  thread runBalayage():
    while (True):
        global ctrl_frequency=350.0
        global weave_frequency=1.2
        global amplitude=0.003
        global cycle_duration=(ctrl_frequency / weave_frequency)
        global pi=3.14159
        global offset=[0.0, 0.0, 0.0, 0.0, 0.0, 0.0]
        global i=0
        path_offset_enable()
        global alpha=0.1
        path_offset_set_alpha_filter(alpha)

        while (True):
          fct_set_offset()
          path_offset_set(offset, 2)
          global i=i+1
          sync()
        end
      end

  end

  def fct_activerBalayage(p_start, p_stop):

      fct_determineAxeBalayage(p_start,p_stop)
      global thr_runBalayage = run runBalayage()

  end

  def fct_desactiverBalayage():

      kill thr_runBalayage

  end
  $ 73 "Script: fcts_ralentir_fin_ligne.script"
  def fct_calcul_point_inter(p_debut,p_fin):

      local p_inter = p_fin

      local poucentage = 0.95
      local inc = 0
      local vecteur_global = p[0,0,0,0,0,0]
      local vecteur_reduit = p[0,0,0,0,0,0]

      while (inc < 6):   #a valider avec d'autres tests (peut etre faire une moyenne)
          vecteur_global[inc] = p_fin[inc] - p_debut[inc]
          vecteur_reduit[inc] = vecteur_global[inc]*poucentage
          p_inter[inc] = p_debut[inc] + vecteur_reduit[inc]
          inc = inc +1
      end

      return p_inter
    end


  $ 351 "Thread_1"
  thread Thread_1():
    while (True):
      $ 352 "Test_Ordre_Marche"
      $ 353 "If Test_Ordre_Mar≟ True "
      if (Test_Ordre_Mar ==   True  ):
        $ 354 "If config_d ≟ 1  or  config_g ≟ 1"
        if (config_d  ==  1   or   config_g  ==  1):
          $ 355 "Set Ordre_Marche=On"
          set_standard_digital_out(0, True)
          $ 356 "Wait: 0.5"
          sleep(0.5)
          $ 357 "If Reponse_Ordre≟ False "
          if (get_standard_digital_in(4) ==   False  ):
            $ 358 "'Si aucune reponse n'a etait recue, arret du programme'"
            # 'Si aucune reponse n'a etait recue, arret du programme'
            $ 359 "close_popup()"
            close_popup()
            $ 360 "Popup: Defaut : L'Ordre marche a ete coupe ( le poste est peu-etre eteint ) "
            popup("Defaut : L'Ordre marche a ete coupe ( le poste est peu-etre eteint ) ", "Error", False, True, blocking=False)
            halt
          end
          $ 361 "Test_Ordre_Mar≔ False "
          global Test_Ordre_Mar=  False
          $ 362 "sync()"
          sync()
        end
      end
      $ 363 "Erreur ordre marche pendant utilisation"
      $ 364 "If Arc_On≟ True   and Reponse_Arc≟ True  and Reponse_Ordre≟ False "
      if (get_standard_digital_out(1) ==   True     and  get_standard_digital_in(5) ==   True    and  get_standard_digital_in(4) ==   False  ):
        $ 365 "'Test pour savoir si ordre marche a ete coupe pendant utilisation'"
        # 'Test pour savoir si ordre marche a ete coupe pendant utilisation'
        $ 366 "close_popup()"
        close_popup()
        $ 367 "Popup: Defaut : Mise sous puissance coupee pendant la trajectoire"
        popup("Defaut : Mise sous puissance coupee pendant la trajectoire", "Error", False, True, blocking=False)
        halt
      end
      $ 368 "sync()"
      sync()
    end
  end
  threadId_Thread_1 = run Thread_1()
  $ 369 "Thread_2"
  thread Thread_2():
    while (True):
      $ 370 "mode_soudure"
      $ 371 "If Mode_soudure ≟  True "
      if (get_configurable_digital_in(3)  ==    True  ):
        $ 372 "If Mode_soudure≟ True  and soudure_on ≟ True "
        if (get_configurable_digital_in(3) ==   True    and  soudure_on  ==   True  ):
          $ 373 "fin_soud≔0"
          global fin_soud=0
          $ 374 "Test_Ordre_Mar≔ True "
          global Test_Ordre_Mar=  True
          $ 375 "Test_Job≔ True "
          global Test_Job=  True
          $ 376 "Wait Test_Ordre_Mar≟ False "
          while (not(Test_Ordre_Mar ==   False  )):
            sync()
          end
          $ 377 "Wait Test_Job≟ False "
          while (not(Test_Job ==   False  )):
            sync()
          end
          $ 378 "Set Arc_On=On"
          set_standard_digital_out(1, True)
          $ 379 "Test_Gaz≔ True "
          global Test_Gaz=  True
          $ 380 "'Test_Gaz permet de faire un appel dans le thread pour tester l'arriver gaz'"
          # 'Test_Gaz permet de faire un appel dans le thread pour tester l'arriver gaz'
          $ 381 "Wait Valide_Gaz≟ True "
          while (not(Valide_Gaz ==   True  )):
            sync()
          end
          $ 382 "'Valide_Gaz permet  de connaitre quand le traitement de l'arriver gaz est terminer ans le thread.'"
          # 'Valide_Gaz permet  de connaitre quand le traitement de l'arriver gaz est terminer ans le thread.'
        else:
          $ 383 "ElseIf Mode_soudure ≟ True  and soudure_on ≟ False "
          if (get_configurable_digital_in(3)  ==   True    and  soudure_on  ==   False  ):
            $ 384 "'Attente post debit gaz'"
            # 'Attente post debit gaz'
            $ 385 "Set Arc_On=Off"
            set_standard_digital_out(1, False)
            $ 386 "Test_Gaz≔ False "
            global Test_Gaz=  False
            $ 387 "Loop Reponse_Arc ≟ 1"
            while (get_standard_digital_in(5)  ==  1):
              $ 388 "fin_soud≔0"
              global fin_soud=0
              $ 389 "sync()"
              sync()
            end
            $ 390 "fin_soud≔1"
            global fin_soud=1
          end
        end
      end
      $ 391 "sync()"
      sync()
    end
  end
  threadId_Thread_2 = run Thread_2()
  $ 392 "Thread_3"
  thread Thread_3():
    while (True):
      $ 393 "led_cobot_2"
      $ 394 "If led_cobot ≟ True "
      if (led_cobot  ==   True  ):
        $ 395 "If valider_bp_co ≟ True "
        if (get_tool_digital_in(0)  ==   True  ):
          $ 396 "Set TO[1]=On"
          set_tool_digital_out(1, True)
          $ 397 "Wait: 0.25"
          sleep(0.25)
          $ 398 "Set TO[1]=Off"
          set_tool_digital_out(1, False)
          $ 399 "Wait: 0.25"
          sleep(0.25)
          $ 400 "Set TO[1]=On"
          set_tool_digital_out(1, True)
          $ 401 "Wait: 0.25"
          sleep(0.25)
          $ 402 "Set TO[1]=Off"
          set_tool_digital_out(1, False)
          $ 403 "Wait: 0.25"
          sleep(0.25)
          $ 404 "Set TO[1]=On"
          set_tool_digital_out(1, True)
          $ 405 "Wait: 0.25"
          sleep(0.25)
          $ 406 "Set TO[1]=Off"
          set_tool_digital_out(1, False)
          $ 407 "Wait: 0.25"
          sleep(0.25)
          $ 408 "sync()"
          sync()
        end
        $ 409 "sync()"
        sync()
      end
      $ 410 "sync()"
      sync()
      $ 411 "sync()"
      sync()
    end
  end
  threadId_Thread_3 = run Thread_3()
  $ 412 "Thread_4"
  thread Thread_4():
    while (True):
      $ 413 "led_cobot"
      $ 414 "If led_cobot ≟ True "
      if (led_cobot  ==   True  ):
        $ 415 "Loop led_cobot ≟  True "
        while (led_cobot  ==    True  ):
          $ 416 "Set TO[0]=On"
          set_tool_digital_out(0, True)
          $ 417 "Wait: 0.5"
          sleep(0.5)
          $ 418 "Set TO[0]=Off"
          set_tool_digital_out(0, False)
          $ 419 "Wait: 0.5"
          sleep(0.5)
          $ 420 "sync()"
          sync()
        end
        $ 421 "sync()"
        sync()
      else:
        $ 422 "Else" "noBreak"
        $ 423 "Set TO[0]=Off"
        set_tool_digital_out(0, False)
        $ 424 "Set TO[1]=Off"
        set_tool_digital_out(1, False)
      end
      $ 425 "sync()"
      sync()
    end
  end
  threadId_Thread_4 = run Thread_4()
  $ 426 "Thread_5"
  thread Thread_5():
    while (True):
      $ 427 "Test_Arc_On"
      $ 428 "Erreur gaz pendant utilisation"
      $ 429 "Timer_gaz"
      $ 430 "If Test_Gaz≟ True "
      if (Test_Gaz ==   True  ):
        $ 431 "Wait: 1.0"
        sleep(1.0)
        $ 432 "Loop Reponse_Arc≟ False  and Arc_On≟ True "
        thread Thread_while_432():
          while (True):
            $ 433 "'La boucle permet d'activer le timer et tester deux condition pour les Defaults'"
            # 'La boucle permet d'activer le timer et tester deux condition pour les Defaults'
            $ 434 "timer_ret_gaz: Start"
            timer_ret_gaz_is_counting = True
            $ 435 "If timer_ret_gaz>0.5"
            global thread_flag_435=0
            thread Thread_if_435():
              $ 436 "'Le timer permet de realiser une attente '"
              # 'Le timer permet de realiser une attente '
              $ 437 "close_popup()"
              close_popup()
              $ 438 "Popup: Defaut : Pas de retour flux, stabilisation gaz"
              popup("Defaut : Pas de retour flux, stabilisation gaz", "Error", False, True, blocking=False)
              halt
              thread_flag_435 = 1
            end
            if (timer_ret_gaz>0.5):
              global thread_handler_435=run Thread_if_435()
              while (thread_flag_435 == 0):
                if not(timer_ret_gaz>0.5):
                  kill thread_handler_435
                  thread_flag_435 = 2
                else:
                  sync()
                end
              end
            else:
              thread_flag_435 = 2
            end
            if (thread_flag_435 == 2):
              $ 439 "ElseIf Reponse_Ordre≟ False "
              if (get_standard_digital_in(4) ==   False  ):
                $ 440 "'Cette condition nous permet de pouvoir tout couper ordre marche pendant la boucle.'"
                # 'Cette condition nous permet de pouvoir tout couper ordre marche pendant la boucle.'
                $ 441 "close_popup()"
                close_popup()
                $ 442 "Popup: Defaut : Perte retour de signal, mise sous puissance generateur"
                popup("Defaut : Perte retour de signal, mise sous puissance generateur", "Error", False, True, blocking=False)
                halt
              end
            end
          end
        end
        if (get_standard_digital_in(5) ==   False    and  get_standard_digital_out(1) ==   True  ):
          global thread_handler_432=run Thread_while_432()
          while (get_standard_digital_in(5) ==   False    and  get_standard_digital_out(1) ==   True  ):
            sync()
          end
          kill thread_handler_432
        end
        $ 443 "Valide_Gaz≔ True "
        global Valide_Gaz=  True
        $ 444 "timer_ret_gaz: Reset"
        timer_ret_gaz = 0
      end
      $ 445 "sync()"
      sync()
    end
  end
  threadId_Thread_5 = run Thread_5()
  $ 446 "Thread_6"
  thread Thread_6():
    while (True):
      $ 447 "Test_Job"
      $ 448 "If Test_Job≟ True "
      if (Test_Job ==   True  ):
        $ 452 "Test_Job≔ False "
        global Test_Job=  False
      end
      $ 453 "sync()"
      sync()
    end
  end
  threadId_Thread_6 = run Thread_6()
  $ 454 "Thread_7"
  thread Thread_7():
    while (True):
      $ 455 "secu"
      $ 456 "If SecuGaucheOk ≟  False  and secu_g ≟ 1"
      if (get_configurable_digital_in(4)  ==    False    and  secu_g  ==  1):
        $ 457 "close_popup()"
        close_popup()
        $ 458 "Popup: ATTENTION : Defaut carter !"
        popup("ATTENTION : Defaut carter !", "Error", False, True, blocking=False)
        halt
      else:
        $ 459 "ElseIf SecuDroiteOk ≟ False  and secu_d ≟ 1"
        if (get_configurable_digital_in(5)  ==   False    and  secu_d  ==  1):
          $ 460 "close_popup()"
          close_popup()
          $ 461 "Popup: ATTENTION : Defaut carter !"
          popup("ATTENTION : Defaut carter !", "Error", False, True, blocking=False)
          halt
        end
      end
      $ 462 "sync()"
      sync()
    end
  end
  threadId_Thread_7 = run Thread_7()
  $ 463 "Thread_8"
  thread Thread_8():
    while (True):
      $ 464 "bloq_soud_arret"
      $ 465 "If Mode_soudure≟ False  and Test_Gaz ≟ True "
      if (get_configurable_digital_in(3) ==   False    and  Test_Gaz  ==   True  ):
        $ 466 "close_popup()"
        close_popup()
        $ 467 "Popup: Defaut : L'ordre de soudure a ete coupe pendant l'utilisation."
        popup("Defaut : L'ordre de soudure a ete coupe pendant l'utilisation.", "Error", False, True, blocking=False)
        halt
      end
      $ 474 "sync()"
      sync()
    end
  end
  threadId_Thread_8 = run Thread_8()
  $ 485 "Thread_10"
  thread Thread_10():
    while (True):
      $ 486 "reglage"
      $ 487 "If safe_mode ≟ 1  and Mode_manu ≟  True "
      if (safe_mode  ==  1   and  get_configurable_digital_in(7)  ==    True  ):
        $ 488 "close_popup()"
        close_popup()
        $ 489 "Popup: STOP !!!!"
        popup("STOP !!!!", "Error", False, True, blocking=False)
        halt
      end
      $ 490 "sync()"
      sync()
      $ 491 "sync()"
      sync()
    end
  end
  threadId_Thread_10 = run Thread_10()
  $ 74 "Robot Program"
  $ 78 "Script: general.script"
  while (True):
    # 68 "Programme de robot"
    global safe_mode=0

    set_configurable_digital_out(0, False)

    set_configurable_digital_out(1, False)

    while (get_configurable_digital_in(4) ==   True    or  get_configurable_digital_in(5) ==   True  ):

      sync()
      # 94 "'clingottement pour signifier qu'il y  un defaut sur un des carters '"
      set_standard_digital_out(4, False)
      set_configurable_digital_out(6, False)
      sleep(0.5)
      set_standard_digital_out(4, True)
      set_configurable_digital_out(6, True)
      sleep(0.5)
      sync()
    end

    set_configurable_digital_out(6, False)
    set_standard_digital_out(4, False)
    sleep(2.0)
    #movel(pose_add(get_target_tcp_pose(), pose_sub(PointPassage_12_to_p, PointPassage_12_from_p)), a=0.01, v=2.0E-4)
    global angle_base= get_actual_joint_positions ()
    if (angle_base[0]  <= 0.7):
      if (angle_base[0] >= 1.6):
        # 116 "Départ"        A CHANGER PAR UNE POSTION ENREGISTREE
        movej([0.7376820445060732, 1.3357652919721463, -2.8533326461405863, -0.44459326684985356, 1.9245067834854124, 4.003490924835204], a=1.3962634015954636, v=1.0471975511965976)
      else:
        if (angle_base[0]>1.6):
          movej(Point_init_D, a=1.3962634015954636, v=1.7453292519943295)
          movej(Point_avt_initD, a=1.3962634015954636, v=1.7453292519943295)
        else:
          if (angle_base[0]<0.7):
            movej(Point_init_G, a=1.3962634015954636, v=1.7453292519943295)
          end
        end
      end
    else:
      # 124 "SinonSi angle_base[0]>1.6"
      if (angle_base[0]>1.6):

        movej(Point_init_D, a=1.3962634015954636, v=1.7453292519943295)
        movej(Point_avt_initD, a=1.3962634015954636, v=1.7453292519943295)
      else:
        if (angle_base[0]<0.7):
          movej(Point_init_G, a=1.3962634015954636, v=1.7453292519943295)
        end
      end
    end
    # 131 "Départ"             A CHANGER PAR UNE POSTION ENREGISTREE
    movej([0.7376820445060732, 1.3357652919721463, -2.8533326461405863, -0.44459326684985356, 1.9245067834854124, 4.003490924835204], a=1.3962634015954636, v=1.0471975511965976)
    global angle_base= get_actual_joint_positions ()
    # 'mode config'
    if (get_configurable_digital_in(7)  ==   False    and  get_standard_digital_in(7)  ==   False  ):
      if ((config_g  ==  1)   and   (config_d  ==  1)):
        pop_up_config_g_et_d()
      else:
        if ((config_g  == 1)):
          pop_up_config_g()
        else:
          if (config_d  ==  1):
            pop_up_config_d()
          else:
            if ((config_g  ==  0)  and  (config_d  ==  0)):
              pop_up_config()
            end
          end
        end
      end
      global boucle=1
      while ((get_configurable_digital_in(7)  ==   False  )  and  (boucle  ==  1)   and  (get_standard_digital_in(7) ==   False  )):
        thread Thread_while_145():
          while (True):
            set_standard_digital_out(5, True)
            set_standard_digital_out(6, False)
            sleep(0.5)
            set_standard_digital_out(5, False)
            set_standard_digital_out(6, True)
            sleep(0.5)
            sync()
          end
        end
        if (get_standard_digital_in(3) ==   False    and  get_standard_digital_in(2) ==   False    and  get_configurable_digital_in(7)  ==    False    and  get_standard_digital_in(7) ==   False  ):
          global thread_handler_145=run Thread_while_145()
          while (get_standard_digital_in(3) ==   False    and  get_standard_digital_in(2) ==   False    and  get_configurable_digital_in(7)  ==    False    and  get_standard_digital_in(7) ==   False  ):
            sync()
          end
          kill thread_handler_145
        end
        if (get_standard_digital_in(2)  ==   True  ):
          set_standard_digital_out(5, True)
          set_standard_digital_out(6, False)
          movej(Point_init_G, a=1.3962634015954636, v=1.0471975511965976, r=0.006)
          movej(Point_Attente_G, a=1.3962634015954636, v=1.0471975511965976, r=0.006)
          movej(Point_config_g, a=0.6981317007977318, v=0.5235987755982988)
          global led_cobot=1
          fun_config_g()
          global led_cobot=0
          fun_valid_config_g()
          movej(Point_Attente_G, a=1.3962634015954636, v=1.0471975511965976, r=0.006)
          movej(Point_init_G, a=1.3962634015954636, v=1.0471975511965976, r=0.006)
          # 170 "Départ"         A CHANGER PAR UNE POSTION ENREGISTREE
          movej([0.7376820445060732, 1.3357652919721463, -2.8533326461405863, -0.44459326684985356, 1.9245067834854124, 4.003490924835204], a=1.3962634015954636, v=1.0471975511965976)
        end

        if (get_standard_digital_in(3)  ==   True  ):
          set_standard_digital_out(6, True)
          set_standard_digital_out(5, False)
          movej(Point_avt_initD, a=1.3962634015954636, v=1.0471975511965976, r=0.006)
          movej(Point_init_D, a=1.3962634015954636, v=1.0471975511965976)
          movej(Point_Attente_D, a=1.3962634015954636, v=1.0471975511965976, r=0.006)
          movej(Point_config_d, a=0.6981317007977318, v=0.5235987755982988)
          global led_cobot=1
          fun_config_d()
          global led_cobot=0
          fun_valid_config_d()
          movej(Point_Attente_D, a=1.3962634015954636, v=1.0471975511965976, r=0.006)
          movej(Point_init_D, a=1.3962634015954636, v=1.0471975511965976, r=0.006)
          movej(Point_avt_initD, a=1.3962634015954636, v=1.0471975511965976, r=0.006)
          # 190 "Départ"         A CHANGER PAR UNE POSTION ENREGISTREE
          movej([0.7376820445060732, 1.3357652919721463, -2.8533326461405863, -0.44459326684985356, 1.9245067834854124, 4.003490924835204], a=1.3962634015954636, v=1.0471975511965976)
        end
      end
    end
    # '"Reglage"'

    if (get_configurable_digital_in(7)  ==   False    and  get_standard_digital_in(7)  ==   True  ):
      if ((config_g  ==  1)   and   (config_d  ==  1)):
        pop_up_reg_gd()
        global boucle=1
      else:
        if (config_g  ==  1):
          pop_up_reg_gd()
          global boucle=1
        else:
          if (config_d  ==  1):
            pop_up_reg_d()
            global boucle=1
          else:
            close_popup()
            while (get_standard_digital_in(7)  ==   True  ):
              popup("Aucune configuration n'est actuellement detectée.", "Erreur", False, True, blocking=True)
            end
          end
        end
      end
      global boucle=1
      while ((get_configurable_digital_in(7)  ==   False  )  and  (boucle  ==  1)   and  (get_standard_digital_in(7) ==   True  )):
        thread Thread_while_208():
          while (True):
            if (config_g  ==  1):
              set_standard_digital_out(5, True)
            end
            if (config_d  ==  1):
              set_standard_digital_out(6, True)
            end
            sleep(0.5)
            set_standard_digital_out(5, False)
            set_standard_digital_out(6, False)
            sleep(0.5)
          end
        end
        if (get_standard_digital_in(3) ==   False    and  get_standard_digital_in(2) ==   False    and  get_configurable_digital_in(7)  ==    False    and  get_standard_digital_in(7)  ==   True  ):
          global thread_handler_208=run Thread_while_208()
          while (get_standard_digital_in(3) ==   False    and  get_standard_digital_in(2) ==   False    and  get_configurable_digital_in(7)  ==    False    and  get_standard_digital_in(7)  ==   True  ):
            sync()
          end
          kill thread_handler_208
        end
        if (get_standard_digital_in(2)  ==   True  ):
          global safe_mode=1
          set_standard_digital_out(5, True)
          set_standard_digital_out(6, False)
          movej(Point_init_G, a=1.3962634015954636, v=1.0471975511965976, r=0.006)
          movej(Point_Attente_G, a=1.3962634015954636, v=1.0471975511965976, r=0.006)
          movej(pose_inter_g, a=0.6981317007977318, v=0.5235987755982988)
          global led_cobot=1
          fun_Pas_A_Pas_g()
          global led_cobot=0
          global safe_mode=0
          global boucle=0
        end
        if (get_standard_digital_in(3)  ==   True  ):
          global safe_mode=1
          set_standard_digital_out(6, True)
          set_standard_digital_out(5, False)
          movej(Point_avt_initD, a=1.3962634015954636, v=1.0471975511965976, r=0.006)
          movej(Point_init_D, a=1.3962634015954636, v=1.0471975511965976, r=0.006)
          movej(pose_inter_d, a=0.6981317007977318, v=0.5235987755982988)
          global led_cobot=1
          fun_Pas_A_Pas_d()
          global led_cobot=0
          global safe_mode=0
          global boucle=0
        end
      end
    end
    # 'mode execution'
    if (get_configurable_digital_in(7)  ==   True  ):
      if ((config_g  ==  1)   and   (config_d  ==  1)):
        pop_up_exe()
        global boucle=1
      else:
        if (config_g  ==  1):
          pop_up_exe_g()
          global boucle=1
        else:
          if (config_d  ==  1):
            pop_up_exe_d()
            global boucle=1
          else:
            close_popup()
            while (get_configurable_digital_in(7)  ==   True  ):
              popup("Aucune programmation n'est actuellement detectée, veillez à programmer une pièce avant de vouloir l'éxécuter.", "Erreur", False, True, blocking=True)
            end
          end
        end
      end
      while (( get_configurable_digital_in(7)  ==   True  )   and  (boucle  ==  1)):
        thread Thread_while_259():
          while (True):
            if (config_g  ==  1):
              set_standard_digital_out(5, True)
            end
            if (config_d  ==  1):
              set_standard_digital_out(6, True)
            end
            sleep(0.5)
            set_standard_digital_out(5, False)
            set_standard_digital_out(6, False)
            sleep(0.5)
          end
        end
        if (get_standard_digital_in(3) ==   False    and  get_standard_digital_in(2) ==   False    and  get_configurable_digital_in(7) ==   True  ):
          global thread_handler_259=run Thread_while_259()
          while (get_standard_digital_in(3) ==   False    and  get_standard_digital_in(2) ==   False    and  get_configurable_digital_in(7) ==   True  ):
            sync()
          end
          kill thread_handler_259
        end
        if ((get_standard_digital_in(2)  ==   True  )  and  (config_g  ==   True  )):
          global boucle_g=1
          while (boucle_g  ==  1):
            set_configurable_digital_out(0, True)
            set_standard_digital_out(5, True)
            set_standard_digital_out(6, False)
            sleep(0.25)
            set_standard_digital_out(5, False)
            sleep(0.25)
            if (get_configurable_digital_in(4)  ==    False  ):
              set_standard_digital_out(5, True)
              if (get_configurable_digital_in(4)  ==    False  ):
                close_popup()
                while (get_configurable_digital_in(4) == False):
                  sync()
                end
              end
            end
            if (get_configurable_digital_in(4)  ==    True  ):
              global secu_g=1
              set_standard_digital_out(5, True)
              movej(Point_init_G, a=1.3962634015954636, v=1.0471975511965976, r=0.006)
              fun_execution_g()
              movej(Point_Attente_G, a=1.3962634015954636, v=1.0471975511965976, r=0.006)
              movej(Point_init_G, a=1.3962634015954636, v=1.0471975511965976, r=0.006)
              # 294 "Départ"         A CHANGER PAR UNE POSTION ENREGISTREE
              movej([0.7376820445060732, 1.3357652919721463, -2.8533326461405863, -0.44459326684985356, 1.9245067834854124, 4.003490924835204], a=1.3962634015954636, v=1.0471975511965976)
              set_configurable_digital_out(0, False)
              global secu_g=0
              global boucle_g=0
            end
          end
          global boucle=0
        else:
          if ((get_standard_digital_in(2)  ==   True  )  and  (config_g  ==   False  )):
            close_popup()
            popup("Aucune programmation n'est actuellement detectée sur la table gauche, veillez à programmer une pièce avant de vouloir l'éxécuter.", "Erreur", False, True, blocking=True)
            global boucle=0
          end
        end
        if ((get_standard_digital_in(3)  ==   True  )  and  (config_d  ==   True  )):
          global boucle_d=1
          pop_up_deb_exe_d()
          while (boucle_d  ==  1):
            set_configurable_digital_out(1, True)
            set_standard_digital_out(5, False)
            set_standard_digital_out(6, True)
            sleep(0.25)
            set_standard_digital_out(6, False)
            sleep(0.25)
            if (get_configurable_digital_in(5)  ==    False  ):
              set_standard_digital_out(6, True)
              sleep(6.0)
              if (get_configurable_digital_in(5)  ==    False  ):
                close_popup()
                while (get_configurable_digital_in(5) == False):
                  sync()
                end
              end
            end
            if (get_configurable_digital_in(5)  ==    True  ):
              global secu_d=1
              set_standard_digital_out(6, True)
              movej(Point_avt_initD, a=1.3962634015954636, v=1.0471975511965976)
              fun_execution_d()
              set_configurable_digital_out(1, False)
              global secu_d=0
              global boucle_d=0
            end
          end
          global boucle=0
        else:
          if ((get_standard_digital_in(3)  ==   True  )  and  (config_d  ==   False  )):
            close_popup()
            popup("Aucune programmation n'est actuellement detectée sur la table droite, veillez à programmer une pièce avant de vouloir l'éxécuter.", "Erreur", False, True, blocking=True)
            global boucle=0
          end
        end
      end
    end
  end
  end
end
